// TIA Portal V20 export
TYPE "LWONIK_typeToSafetyDoorSelect"
// stored: Access Published
   STRUCT
      Front_UnwinderMStageDoorSelect : Bool;
      Front_NotchingDoorSelect : Bool;
      Front_VisionDoorSelect : Bool;
      Rear_UnwinderDoorSelect : Bool;
      Rear_NotchingDoorSelect : Bool;
      Rear_VisionDoorSelect : Bool;
      Rear_RewinderDoorSelect : Bool;
      Rear_ScrapCutterSelect : Bool;
      DoorLock : Bool;
      DoorUnlock : Bool;
   END_STRUCT;
END_TYPE
